FUNCTION_BLOCK FB_ContainerDefGrid EXTENDS FB_ContainerBase
VAR_INPUT
END_VAR
VAR_OUTPUT
END_VAR
VAR
  fBImageDeformation : FB_ImageDeformation;
END_VAR

fBImageDeformation();                       // call run cyclic image deformation
fBImageDeformation.LogLevel := LogLevel;    // distribute container logLevel to image deformation fb

METHOD AbortDeformation : BOOL
VAR_INPUT
  sReason   : STRING;
  Src       : REFERENCE TO T_ErrSrc;
  bHideLog  : BOOL;
END_VAR
IF NOT bHideLog THEN
  LogWarning(F_Concat4('Abort deformation: ', sReason, ' Src: ', Src.aDescr));  // log reason
END_IF
setError(ErrDef:=EC_DefGrid.ecDefGrid_DefGridAbort, Src:=Src); // tag ct as error
fBImageDeformation.abort();  // abort deformation
StopScript(iCT:=THIS^);
END_METHOD

METHOD AddCamPoint : BOOL
VAR_INPUT
  sPoint : ST_DeformationPointAccurate;
END_VAR
AddCamPoint := fBImageDeformation.addCamPoint(sNewPoint:=sPoint);
END_METHOD

(*
  Create a container, build very basics.
*)
METHOD Create : BOOL
VAR_INPUT
	nCTId	            : DINT;     (* a container identifier *)
	nCTIndex	        : UDINT;	  (* memory index (array index if CT in CT array) *)
END_VAR
SUPER^.Create(nCTId:=nCTId, nCTIndex:=nCTIndex);
fBImageDeformation.reset();
fBImageDeformation.nProcessId := THIS^.pCT^.iId;
END_METHOD

PROPERTY eCamMode : E_CameraMode
GET
eCamMode := fBImageDeformation.eCamMode;
END_GET
END_PROPERTY

(*
  Shift in x [SubPx]
*)
PROPERTY fDxShift : LREAL
GET
VAR
  errCtr : UDINT;
END_VAR
fDxShift := fBImageDeformation._nDxShift;
END_GET
END_PROPERTY

(*
  Shift in y [Px]
*)
PROPERTY fDyShift : LREAL
GET
VAR
  errCtr : UDINT;
END_VAR
fDyShift := fBImageDeformation._nDyShift;
END_GET
END_PROPERTY

PROPERTY fPrintLengthEffective : LREAL
GET
fPrintLengthEffective := fBImageDeformation.fPrintLengthEffective;
END_GET
END_PROPERTY

(*
  get a deformation point.
  :returns: TRUE if successful
*)
METHOD getDeformationPoint : BOOL;
VAR_INPUT
  nCol : UDINT;   // col select
  nRow : UDINT;   // row select
END_VAR
VAR_OUTPUT
  sPoint : ST_DeformationPointAccurate;
END_VAR
getDeformationPoint := fBImageDeformation.getDeformationPoint(nCol:=nCol, nRow:=nRow, sPoint=>sPoint);
END_METHOD

(*
  Deformation state of CT.
  :return:  TRUE in case of error -> any deformation error
*)
METHOD getDeformationStatus : BOOL
VAR_INPUT
END_VAR
VAR_OUTPUT
  eDStep: E_DeformationStep;// deformation step
  bDone : BOOL;             // deformation done
  bBusy : BOOL;             // deformation is busy
  nErrorId : UDINT;         // error id in case of error
  tExecutionTime : TIME;    // script update execution time?
  bAborted : BOOL;          // deformation is aborted/error
END_VAR
getDeformationStatus := fBImageDeformation.bError;

eDStep:= fBImageDeformation.eStep;
bBusy := fBImageDeformation.bBusy;
bDone := fBImageDeformation.bDone;
nErrorId := fBImageDeformation.nErrorId;
tExecutionTime := fBImageDeformation.tExecutionTime;
bAborted := fBImageDeformation.bAborted;
END_METHOD

PROPERTY nAvailableGridCols : UDINT
GET
nAvailableGridCols := fBImageDeformation._nGridCols;
END_GET
END_PROPERTY

PROPERTY nAvailableGridPoints : UDINT
GET
nAvailableGridPoints := fBImageDeformation.nAvailableGridPoints;
END_GET
END_PROPERTY

PROPERTY PUBLIC nRegisteredCameraPoints : UDINT
GET
nRegisteredCameraPoints := fBImageDeformation._nCamPoints;
END_GET
END_PROPERTY

PROPERTY sDefGridSettings : ST_DefGridSettings
GET
sDefGridSettings := fBImageDeformation.sDefGridSettings;
END_GET
END_PROPERTY

METHOD StartCamera
VAR_INPUT
  eCameraMode  : E_CameraMode;   // used camera mode
  fFeatureGrid : LREAL;          // deformation module update interval [Px]
  bResetDeformation : BOOL;      // reset current deformation state
END_VAR
// reset old deformation
IF bResetDeformation THEN
  fBImageDeformation.reset();
END_IF

// update mode
fBImageDeformation.eCamMode := eCameraMode;
fBImageDeformation.fFeatureGrid := fFeatureGrid;
fBImageDeformation.eStep := E_DeformationStep.cameraStarted;
END_METHOD

METHOD StartDeformation
VAR_INPUT
  sDefGridSettings : ST_DefGridSettings;
  fStartDeformationPos : LREAL;   // reference start position in [px]
END_VAR
fBImageDeformation.fPrintLengthEffective := pJob^.fSubstrateDepth;                           // update with intended length 
fBImageDeformation.sDefGridSettings := sDefGridSettings;                  // apply grid setting
fBImageDeformation.startDeformation(                                      // start deformation process
  fStartDefPos:=fStartDeformationPos     // reference position at current position [Px]
);
END_METHOD

METHOD StartScript
VAR_INPUT
  iDeformationHandler : I_DeformationHandler;
END_VAR
fBImageDeformation.iDeformationHandler := iDeformationHandler;
fBImageDeformation.eStep := E_DeformationStep.createdScriptContainer;
END_METHOD

METHOD StopScript : BOOL
VAR_INPUT
  iCT : I_CT;
END_VAR
IF fBImageDeformation.iDeformationHandler <> 0 THEN
  fBImageDeformation.iDeformationHandler.DeleteCachedCt(iCT:=iCT);
  fBImageDeformation.iDeformationHandler := 0; // remove handler after stopping (prevent further calls on same CT)
END_IF
END_METHOD

METHOD UpdateDeformation
VAR_INPUT
  fPos : LREAL; // relative deformation position in [px]
END_VAR
fBImageDeformation.updateDeformation(fPos:=fPos);
END_METHOD

END_FUNCTION_BLOCK

(* stored: Version 1.1.0.1, ProductVersion 3.1.4024.11
   POU FB_ContainerDefGrid: Id {2d8beb5a-7741-4f53-9b5d-5bba1cb243c4}, SpecialFunc None
   Method AbortDeformation: Id {f4e769e7-fdcb-497a-869a-11c396829281}
   Method AddCamPoint: Id {c9a7845c-22a0-4577-acbe-8954df2e199f}
   Method Create: Id {e7db097f-b805-4a15-997e-aea4a4252e85}
   Property eCamMode: Id {908be121-4ce8-47bc-b894-67ea1d9badcb}
   Get Get: Id {4771b49c-2100-4b65-8c92-af55ada05f98}
   Property fDxShift: Id {f4b62b6e-2ae9-4fbc-b999-716d94294e90}
   Get Get: Id {66c9eb50-0679-4295-8ac5-c47a55b9a9c4}
   Property fDyShift: Id {a1bfccb0-2d05-4dbc-897b-c5caf07669b4}
   Get Get: Id {1d2c50e2-c63a-41c7-9fdd-72e3032bf798}
   Property fPrintLengthEffective: Id {fc4e2877-6a77-41c5-8f15-21a5e29b64d2}
   Get Get: Id {3635365e-9f81-49d8-b457-62cabb39356f}
   Method getDeformationPoint: Id {2c7c8e7c-37b2-43e1-90a8-ea784d68621e}
   Method getDeformationStatus: Id {ad3cfac4-eda3-4d41-892b-ffdca204925e}
   Property nAvailableGridCols: Id {61be60fa-e3b9-4821-925e-23b920d7bfd3}
   Get Get: Id {8f97e19b-db85-4e14-95e2-7bc242c47118}
   Property nAvailableGridPoints: Id {d70e9fbe-44b3-4e41-aa7d-d45874a9762c}
   Get Get: Id {a3e9e991-2e2d-4b0b-9b38-b97f16ba20be}
   Property nRegisteredCameraPoints: Id {f813e15a-dac8-4907-83e3-431c7dfe5c84}
   Get Get: Id {e0059d97-ca3c-4ec0-8b56-5e7d4cb3596c}
   Property sDefGridSettings: Id {f9976eb4-29cd-4f5b-9829-bbe8c23a9ab1}
   Get Get: Id {bebda86e-82b9-4a1b-b7e5-739d4c134a65}
   Method StartCamera: Id {fa9cfc27-a9f9-4b08-a02d-72b82e2069db}
   Method StartDeformation: Id {9e341afe-e643-4f6d-8b0c-fa3d83df99bb}
   Method StartScript: Id {b42a5bf2-aedf-44f3-9b19-80a8065b52ca}
   Method StopScript: Id {eb4b604b-26be-4db7-b553-a71f9287a6bd}
   Method UpdateDeformation: Id {ca2f28fa-632e-448d-aace-7cab62296cdd} *)
